% RSLogix 500 project Q4.RSS, saved by version 8.30.00.16 %
PROJECT "Q4"    % processor: Bul.1763 MicroLogix 1100 Series B %

PROGRAM FILES
  LAD 2   4 rungs

DATA FILES
  O0 OUTPUT  4 elements
  I1 INPUT  6 elements
  S2 STATUS  66 elements
  B3 BINARY  1 elements
  T4 TIMER  1 elements
  C5 COUNTER  1 elements
  R6 CONTROL  1 elements
  N7 INTEGER  1 elements
  F8 FLOAT  1 elements

LADDER 2
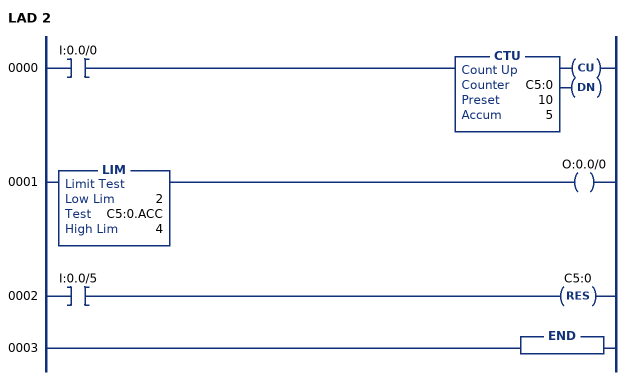
% Rung: 0 %
SOR XIC I:0.0/0 CTU C5:0 10 5 EOR
% Rung: 1 %
SOR LIM 2 C5:0.ACC 4 OTE O:0.0/0 EOR
% Rung: 2 %
SOR XIC I:0.0/5 RES C5:0 EOR
% Rung: 3 %
SOR END EOR

OTHER DOCUMENTED ADDRESSES
  O:0.0/2  "lamp"

DATA TABLE (non-zero values as saved)
DATA C5
% .PRE .ACC %
% C5:0 % 10 5
